{attribute addProperty BoxType "EL2535-0000-0016"}
{attribute addProperty Id "PWM_Status_ChannelAT %I*ARRAY[0..1] OF PWM_Status_Channel_BFDF08183240PWM_Control_ChannelAT %Q*ARRAY[0..1] OF PWM_Control_Channel_253BEA616480WcStateAT %I*WcState_98A4DF7520.250InfoDataAT %I*InfoData_BC63D37F80100"}
{attribute addProperty CRC "1732075894"}
{attribute addProperty SizeInBites "178"}
{attribute addProperty SizeInBytes "22.25"}
TYPE EL2535_81CB2727 :
STRUCT
	{attribute addProperty Name "PWM_Status_Channel"}
	PWM_Status_Channel : ARRAY[0..1] OF PWM_Status_Channel_BFDF0818;
	{attribute addProperty Name "PWM_Control_Channel"}
	PWM_Control_Channel : ARRAY[0..1] OF PWM_Control_Channel_253BEA61;
	{attribute addProperty Name "WcState"}
	WcState : WcState_98A4DF75;
	{attribute addProperty Name "InfoData"}
	InfoData : InfoData_BC63D37F;
END_STRUCT
END_TYPE

(* stored: Version 1.2.0.0, ProductVersion 3.1.4024.9
   DUT EL2535_81CB2727: Id {0184b34c-bbd4-4cdd-8cb4-ff99f6f13da7} *)
